RoboDK station: RK3 extrudy.rdk

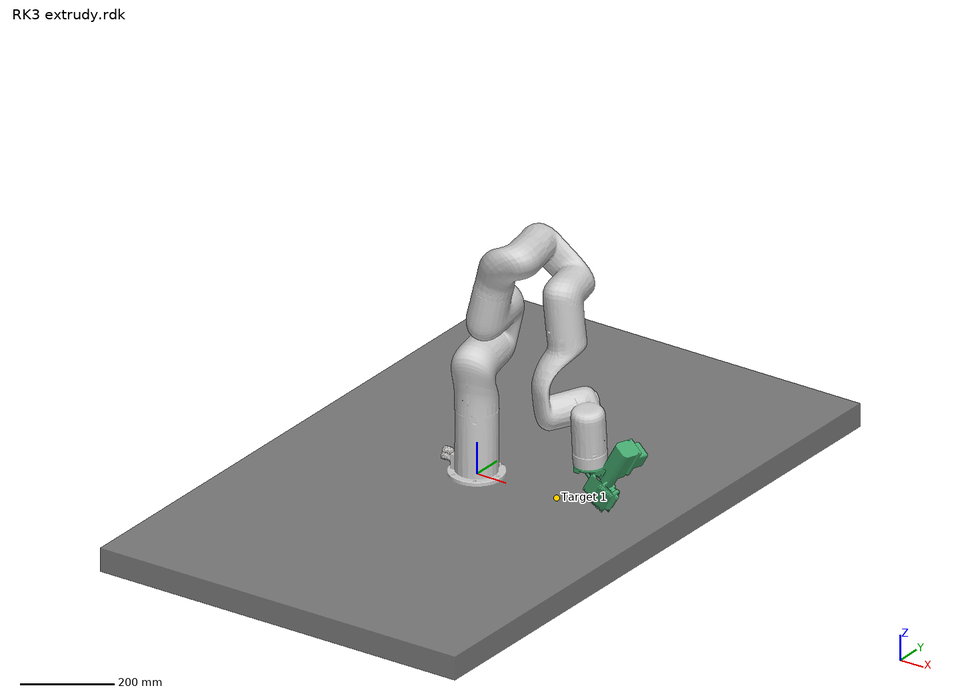
[picture v0: the station drawn from its stored meshes, robots at their saved joint values, targets as dots, program paths as lines]
Station RK3 extrudy (saved by RoboDK 5.5.0). Poses are relative to the parent item; angles as X-Y-Z fixed-axis rotations.
Station parameters (name, value as stored): CollisionFreePlanner, uFactory xArm6 11-16-2023 clayextruder, CollisionFreePlanner-Rob uFactory xArm6 11-16-2023 clayextruder
  - frame uFactory xArm6 Base at (0, 1000, 0) mm
    - robot uFactory xArm6 11-16-2023 clayextruder (model uFactory xArm6): 6 axes, payload 5 kg, reach 700 mm, repeatability 0.1 mm, weight 12.2 kg
        modified DH rows (alpha deg, a mm, theta deg, d mm): 0, 0, 0, 267; -90, 0, -79.35, 0; 0, 289.489, 79.35, 0; -90, 77.5, 0, 342.5; 90, 0, 0, 0; -90, 76, 0, 97
        joint limits [-360, -118, -225, -360, -81, -124] to [360, 120, 11, 360, 180, 110]; home [0, 0, 0, 0, 0, 0]; saved at [11.871, 11.935, -17.899, 43.294, 7.272, -31.184]
      - tool WASP extruder, TCP at (0, 0, 108) mm, rotated rx 0 ry -30.3 rz 0 deg, size 160.2 x 105.1 x 183.1 mm, geometry from uFactory xArm6 Base
  - frame uFactory xArm6 Base at (0, 1000, 0) mm
    - object table at (0, 0, 0) mm, rotated rx 90 ry 0 rz 90 deg, size 1500 x 55 x 920 mm, geometry from table.obj
    - target Target 1 (Cartesian target) at (207, 0, 0.5) mm, rotated rx -180 ry 30.3 rz 0 deg; joints [0, 0, 0, 0, 0, 0] of uFactory xArm6 11-16-2023 clayextruder
  - Python program Prog2 (listed below)

--- Python program Prog2 ---
# Type help("robodk.robolink") or help("robodk.robomath") for more information
# Press F5 to run the script
# Documentation: https://robodk.com/doc/en/RoboDK-API.html
# Reference:     https://robodk.com/doc/en/PythonAPI/robodk.html
# Note: It is not required to keep a copy of this file, your Python script is saved with your RDK project

# Forward and backwards compatible use of the RoboDK API:
# Remove these 2 lines to follow python programming guidelines
from robodk import *      # RoboDK API
from robolink import *    # Robot toolbox
# Link to RoboDK
# RDK = Robolink()

#generated with Grasshopper for Rhino
#Chris Morrey

import os
import sys
import time
import math

sys.path.append("C:\\Users\\morr0289\\Documents\\Github\\RobotArm\\Python\\")

from arm_sdk3.xarm.wrapper.xarm_api import XArmAPI
arm = XArmAPI('192.168.1.240')
id = 9
baudRate = 9600

if arm.warn_code != 0:
    arm.clean_warn()
if arm.error_code != 0:
    arm.clean_error()
time.sleep(2)

ret = arm.core.set_modbus_timeout(7)
print('set modbus timeout, ret = %d' % (ret[0]))
ret = arm.core.set_modbus_baudrate(baudRate)
print('set modbus baudrate, ret = %d' % (ret[0]))

time.sleep(1)
line = 102

def errors(returned):
    if returned == 1:
        print('1: uncleared error exists')
    elif returned == 23:
        print('23:modbus reply length error')
    elif returned == 20:
        print('20: wrong slave id')
    elif returned == 15:
        print('15: Modbus commands full')
    elif returned == 19:
        print('19: communication error')
    elif returned == 28:
        print('28: end module communication error')
    else:
        print('other error: ',returned)
    input=('clear errors? (y/n)')
    if input == 'y':
            arm.clean_error()
    else:
        print('error not cleared; quitting...')
        time.sleep(2)
        quit()
def sender(data_frame):
    global line
    global id
    #arm.clean_error()
    arm.set_state(state=0)
    code, digitals = arm.get_tgpio_digital()
    #while arm.connected and arm.error_code != 19 and arm.error_code != 28:
    if code == 0 and digitals[0] == 1:
        print ('extruder reports ready')
        ret = arm.getset_tgpio_modbus_data(data_frame,host_id=id)
        if ret[0] == 0:
            print('wrote ',data_frame[8],data_frame[9],data_frame[10])
            print('got back this: ',ret[1])
            print('line: ',line)
            line += 3
            time.sleep(.75)
    elif digitals [0] == 0:
        print('extruder reports not ready')
    elif code != 0:
        errors(ret[0])

arm.motion_enable(enable=True)
arm.set_mode(0)
arm.set_state(state=0)

arm.set_tcp_load(weight=0.91, center_of_gravity=[0,80,-40])
arm.set_tcp_offset([0,0,110,0,30.3,0], is_radian=False)
arm.set_collision_tool_model(22, x=40, y=40, z=110)

last_digitals = [-1, -1]

'''TGPIO for air solenoid---------------------------------------------
value = 0

    code = arm.set_cgpio_digital_output_function(i, value)
    print('set_cgpio_digital_output_function({}, {}), code={}'.format(i, value, code))
# Reset: 255
for i in range(4, 8):
    code = arm.set_cgpio_digital_output_function(i, 255)
    print('set_cgpio_digital_output_function({}, {}), code={}'.format(i, value, code))'''


arm.reset(wait=True)
if arm.warn_code != 0:
    arm.clean_warn()
if arm.error_code != 0:
    arm.clean_error()

while arm.connected and arm.error_code == 0:
#data is big-endian
    arm.set_position(x=272.50, y=-10.76, z=1.85, roll=180.0, pitch=-30.0, yaw=0.00, speed=30.00, is_radian=False, wait=True)
    datas = [0x09,0x10,0x00,0x00,0x00,0x04,0x08,0x00,0x15,0x00,0x06,0x00,0x01,0x00,0x65]
    sender(datas)
    arm.set_position(x=272.50, y=10.76, z=1.85, roll=180.0, pitch=-30.0, yaw=0.00, speed=30.00, is_radian=False, wait=True)
    datas = [0x09,0x10,0x00,0x00,0x00,0x04,0x08,0x00,0x05,0x00,0x06,0x00,0x01,0x00,0x68]
    sender(datas)
    arm.set_position(x=275.05, y=15.69, z=1.85, roll=180.0, pitch=-30.0, yaw=0.00, speed=30.00, is_radian=False, wait=True)
    datas = [0x09,0x10,0x00,0x00,0x00,0x04,0x08,0x00,0x1f,0x00,0x06,0x00,0x01,0x00,0x6b]
    sender(datas)
    arm.set_position(x=275.05, y=-15.69, z=1.85, roll=180.0, pitch=-30.0, yaw=0.00, speed=30.00, is_radian=False, wait=True)
    datas = [0x09,0x10,0x00,0x00,0x00,0x04,0x08,0x00,0x04,0x00,0x06,0x00,0x01,0x00,0x6e]
    sender(datas)
    arm.set_position(x=277.60, y=-19.35, z=1.85, roll=180.0, pitch=-30.0, yaw=0.00, speed=30.00, is_radian=False, wait=True)
    datas = [0x09,0x10,0x00,0x00,0x00,0x04,0x08,0x00,0x26,0x00,0x06,0x00,0x01,0x00,0x71]
    sender(datas)
    arm.set_position(x=277.60, y=19.35, z=1.85, roll=180.0, pitch=-30.0, yaw=0.00, speed=30.00, is_radian=False, wait=True)
    datas = [0x09,0x10,0x00,0x00,0x00,0x04,0x08,0x00,0x03,0x00,0x06,0x00,0x01,0x00,0x74]
    sender(datas)
    arm.set_position(x=280.15, y=22.36, z=1.85, roll=180.0, pitch=-30.0, yaw=0.00, speed=30.00, is_radian=False, wait=True)
    datas = [0x09,0x10,0x00,0x00,0x00,0x04,0x08,0x00,0x2c,0x00,0x06,0x00,0x01,0x00,0x77]
    sender(datas)
    arm.set_position(x=280.15, y=-22.36, z=1.85, roll=180.0, pitch=-30.0, yaw=0.00, speed=30.00, is_radian=False, wait=True)
    datas = [0x09,0x10,0x00,0x00,0x00,0x04,0x08,0x00,0x03,0x00,0x06,0x00,0x01,0x00,0x7a]
    sender(datas)
    arm.set_position(x=282.70, y=-24.96, z=1.85, roll=180.0, pitch=-30.0, yaw=0.00, speed=30.00, is_radian=False, wait=True)
    datas = [0x09,0x10,0x00,0x00,0x00,0x04,0x08,0x00,0x31,0x00,0x06,0x00,0x01,0x00,0x7d]
    sender(datas)
    arm.set_position(x=282.70, y=24.96, z=1.85, roll=180.0, pitch=-30.0, yaw=0.00, speed=30.00, is_radian=False, wait=True)
    datas = [0x09,0x10,0x00,0x00,0x00,0x04,0x08,0x00,0x03,0x00,0x06,0x00,0x01,0x00,0x80]
    sender(datas)
    arm.set_position(x=285.25, y=27.27, z=1.85, roll=180.0, pitch=-30.0, yaw=0.00, speed=30.00, is_radian=False, wait=True)
    datas = [0x09,0x10,0x00,0x00,0x00,0x04,0x08,0x00,0x36,0x00,0x06,0x00,0x01,0x00,0x83]
    sender(datas)
    arm.set_position(x=285.25, y=-27.27, z=1.85, roll=180.0, pitch=-30.0, yaw=0.00, speed=30.00, is_radian=False, wait=True)
    datas = [0x09,0x10,0x00,0x00,0x00,0x04,0x08,0x00,0x03,0x00,0x06,0x00,0x01,0x00,0x86]
    sender(datas)
    arm.set_position(x=287.80, y=-29.36, z=1.85, roll=180.0, pitch=-30.0, yaw=0.00, speed=30.00, is_radian=False, wait=True)
    datas = [0x09,0x10,0x00,0x00,0x00,0x04,0x08,0x00,0x3a,0x00,0x06,0x00,0x01,0x00,0x89]
    sender(datas)
    arm.set_position(x=287.80, y=29.36, z=1.85, roll=180.0, pitch=-30.0, yaw=0.00, speed=30.00, is_radian=False, wait=True)
    datas = [0x09,0x10,0x00,0x00,0x00,0x04,0x08,0x00,0x03,0x00,0x06,0x00,0x01,0x00,0x8c]
    sender(datas)
    arm.set_position(x=290.35, y=31.27, z=1.85, roll=180.0, pitch=-30.0, yaw=0.00, speed=30.00, is_radian=False, wait=True)
    datas = [0x09,0x10,0x00,0x00,0x00,0x04,0x08,0x00,0x3e,0x00,0x06,0x00,0x01,0x00,0x8f]
    sender(datas)
    arm.set_position(x=290.35, y=-31.27, z=1.85, roll=180.0, pitch=-30.0, yaw=0.00, speed=30.00, is_radian=False, wait=True)
    datas = [0x09,0x10,0x00,0x00,0x00,0x04,0x08,0x00,0x03,0x00,0x06,0x00,0x01,0x00,0x92]
    sender(datas)
    arm.set_position(x=292.90, y=-33.03, z=1.85, roll=180.0, pitch=-30.0, yaw=0.00, speed=30.00, is_radian=False, wait=True)
    datas = [0x09,0x10,0x00,0x00,0x00,0x04,0x08,0x00,0x42,0x00,0x06,0x00,0x01,0x00,0x95]
    sender(datas)
    arm.set_position(x=292.90, y=33.03, z=1.85, roll=180.0, pitch=-30.0, yaw=0.00, speed=30.00, is_radian=False, wait=True)
    datas = [0x09,0x10,0x00,0x00,0x00,0x04,0x08,0x00,0x03,0x00,0x06,0x00,0x01,0x00,0x98]
    sender(datas)
    arm.set_position(x=295.45, y=34.66, z=1.85, roll=180.0, pitch=-30.0, yaw=0.00, speed=30.00, is_radian=False, wait=True)
    datas = [0x09,0x10,0x00,0x00,0x00,0x04,0x08,0x00,0x45,0x00,0x06,0x00,0x01,0x00,0x9b]
    sender(datas)
    arm.set_position(x=295.45, y=-34.66, z=1.85, roll=180.0, pitch=-30.0, yaw=0.00, speed=30.00, is_radian=False, wait=True)
    datas = [0x09,0x10,0x00,0x00,0x00,0x04,0x08,0x00,0x02,0x00,0x06,0x00,0x01,0x00,0x9e]
    sender(datas)
    arm.set_position(x=298.00, y=-36.18, z=1.85, roll=180.0, pitch=-30.0, yaw=0.00, speed=30.00, is_radian=False, wait=True)
    datas = [0x09,0x10,0x00,0x00,0x00,0x04,0x08,0x00,0x48,0x00,0x06,0x00,0x01,0x00,0xa1]
    sender(datas)
    arm.set_position(x=298.00, y=36.18, z=1.85, roll=180.0, pitch=-30.0, yaw=0.00, speed=30.00, is_radian=False, wait=True)
    datas = [0x09,0x10,0x00,0x00,0x00,0x04,0x08,0x00,0x02,0x00,0x06,0x00,0x01,0x00,0xa4]
    sender(datas)
    arm.set_position(x=300.55, y=37.60, z=1.85, roll=180.0, pitch=-30.0, yaw=0.00, speed=30.00, is_radian=False, wait=True)
    datas = [0x09,0x10,0x00,0x00,0x00,0x04,0x08,0x00,0x4b,0x00,0x06,0x00,0x01,0x00,0xa7]
    sender(datas)
    arm.set_position(x=300.55, y=-37.60, z=1.85, roll=180.0, pitch=-30.0, yaw=0.00, speed=30.00, is_radian=False, wait=True)
    datas = [0x09,0x10,0x00,0x00,0x00,0x04,0x08,0x00,0x02,0x00,0x06,0x00,0x01,0x00,0xaa]
    sender(datas)
    arm.set_position(x=303.10, y=-38.95, z=1.85, roll=180.0, pitch=-30.0, yaw=0.00, speed=30.00, is_radian=False, wait=True)
    datas = [0x09,0x10,0x00,0x00,0x00,0x04,0x08,0x00,0x4d,0x00,0x06,0x00,0x01,0x00,0xad]
    sender(datas)
    arm.set_position(x=303.10, y=38.95, z=1.85, roll=180.0, pitch=-30.0, yaw=0.00, speed=30.00, is_radian=False, wait=True)
    datas = [0x09,0x10,0x00,0x00,0x00,0x04,0x08,0x00,0x02,0x00,0x06,0x00,0x01,0x00,0xb0]
    sender(datas)
    arm.set_position(x=305.65, y=40.21, z=1.85, roll=180.0, pitch=-30.0, yaw=0.00, speed=30.00, is_radian=False, wait=True)
    datas = [0x09,0x10,0x00,0x00,0x00,0x04,0x08,0x00,0x50,0x00,0x06,0x00,0x01,0x00,0xb3]
    sender(datas)
    arm.set_position(x=305.65, y=-40.21, z=1.85, roll=180.0, pitch=-30.0, yaw=0.00, speed=30.00, is_radian=False, wait=True)
    datas = [0x09,0x10,0x00,0x00,0x00,0x04,0x08,0x00,0x02,0x00,0x06,0x00,0x01,0x00,0xb6]
    sender(datas)
    arm.set_position(x=308.20, y=-41.40, z=1.85, roll=180.0, pitch=-30.0, yaw=0.00, speed=30.00, is_radian=False, wait=True)
    datas = [0x09,0x10,0x00,0x00,0x00,0x04,0x08,0x00,0x52,0x00,0x06,0x00,0x01,0x00,0xb9]
    sender(datas)
    arm.set_position(x=308.20, y=41.40, z=1.85, roll=180.0, pitch=-30.0, yaw=0.00, speed=30.00, is_radian=False, wait=True)
    datas = [0x09,0x10,0x00,0x00,0x00,0x04,0x08,0x00,0x02,0x00,0x06,0x00,0x01,0x00,0xbc]
    sender(datas)
    arm.set_position(x=310.75, y=42.53, z=1.85, roll=180.0, pitch=-30.0, yaw=0.00, speed=30.00, is_radian=False, wait=True)
    datas = [0x09,0x10,0x00,0x00,0x00,0x04,0x08,0x00,0x55,0x00,0x06,0x00,0x01,0x00,0xbf]
    sender(datas)
    arm.set_position(x=310.75, y=-42.53, z=1.85, roll=180.0, pitch=-30.0, yaw=0.00, speed=30.00, is_radian=False, wait=True)
    datas = [0x09,0x10,0x00,0x00,0x00,0x04,0x08,0x00,0x02,0x00,0x06,0x00,0x01,0x00,0xc2]
    sender(datas)
    arm.set_position(x=313.30, y=-43.60, z=1.85, roll=180.0, pitch=-30.0, yaw=0.00, speed=30.00, is_radian=False, wait=True)
    datas = [0x09,0x10,0x00,0x00,0x00,0x04,0x08,0x00,0x57,0x00,0x06,0x00,0x01,0x00,0xc5]
    sender(datas)
    arm.set_position(x=313.30, y=43.60, z=1.85, roll=180.0, pitch=-30.0, yaw=0.00, speed=30.00, is_radian=False, wait=True)
    datas = [0x09,0x10,0x00,0x00,0x00,0x04,0x08,0x00,0x02,0x00,0x06,0x00,0x01,0x00,0xc8]
    sender(datas)
    arm.set_position(x=315.85, y=44.62, z=1.85, roll=180.0, pitch=-30.0, yaw=0.00, speed=30.00, is_radian=False, wait=True)
    datas = [0x09,0x10,0x00,0x00,0x00,0x04,0x08,0x00,0x59,0x00,0x06,0x00,0x01,0x00,0xcb]
    sender(datas)
    arm.set_position(x=315.85, y=-44.62, z=1.85, roll=180.0, pitch=-30.0, yaw=0.00, speed=30.00, is_radian=False, wait=True)
    datas = [0x09,0x10,0x00,0x00,0x00,0x04,0x08,0x00,0x02,0x00,0x06,0x00,0x01,0x00,0xce]
    sender(datas)
    arm.set_position(x=318.40, y=-45.58, z=1.85, roll=180.0, pitch=-30.0, yaw=0.00, speed=30.00, is_radian=False, wait=True)
    datas = [0x09,0x10,0x00,0x00,0x00,0x04,0x08,0x00,0x5b,0x00,0x06,0x00,0x01,0x00,0xd1]
    sender(datas)
    arm.set_position(x=318.40, y=45.58, z=1.85, roll=180.0, pitch=-30.0, yaw=0.00, speed=30.00, is_radian=False, wait=True)
    datas = [0x09,0x10,0x00,0x00,0x00,0x04,0x08,0x00,0x02,0x00,0x06,0x00,0x01,0x00,0xd4]
    sender(datas)
    arm.set_position(x=320.95, y=46.49, z=1.85, roll=180.0, pitch=-30.0, yaw=0.00, speed=30.00, is_radian=False, wait=True)
    datas = [0x09,0x10,0x00,0x00,0x00,0x04,0x08,0x00,0x5c,0x00,0x06,0x00,0x01,0x00,0xd7]
    sender(datas)
    arm.set_position(x=320.95, y=-46.49, z=1.85, roll=180.0, pitch=-30.0, yaw=0.00, speed=30.00, is_radian=False, wait=True)
    datas = [0x09,0x10,0x00,0x00,0x00,0x04,0x08,0x00,0x02,0x00,0x06,0x00,0x01,0x00,0xda]
    sender(datas)
    arm.set_position(x=323.50, y=-47.36, z=1.85, roll=180.0, pitch=-30.0, yaw=0.00, speed=30.00, is_radian=False, wait=True)
    datas = [0x09,0x10,0x00,0x00,0x00,0x04,0x08,0x00,0x5e,0x00,0x06,0x00,0x01,0x00,0xdd]
    sender(datas)
    arm.set_position(x=323.50, y=47.36, z=1.85, roll=180.0, pitch=-30.0, yaw=0.00, speed=30.00, is_radian=False, wait=True)
    datas = [0x09,0x10,0x00,0x00,0x00,0x04,0x08,0x00,0x02,0x00,0x06,0x00,0x01,0x00,0xe0]
    sender(datas)
    arm.set_position(x=326.05, y=48.19, z=1.85, roll=180.0, pitch=-30.0, yaw=0.00, speed=30.00, is_radian=False, wait=True)
    datas = [0x09,0x10,0x00,0x00,0x00,0x04,0x08,0x00,0x60,0x00,0x06,0x00,0x01,0x00,0xe3]
    sender(datas)
    arm.set_position(x=326.05, y=-48.19, z=1.85, roll=180.0, pitch=-30.0, yaw=0.00, speed=30.00, is_radian=False, wait=True)
    datas = [0x09,0x10,0x00,0x00,0x00,0x04,0x08,0x00,0x02,0x00,0x06,0x00,0x01,0x00,0xe6]
    sender(datas)
    arm.set_position(x=328.60, y=-48.97, z=1.85, roll=180.0, pitch=-30.0, yaw=0.00, speed=30.00, is_radian=False, wait=True)
    datas = [0x09,0x10,0x00,0x00,0x00,0x04,0x08,0x00,0x61,0x00,0x06,0x00,0x01,0x00,0xe9]
    sender(datas)
    arm.set_position(x=328.60, y=48.97, z=1.85, roll=180.0, pitch=-30.0, yaw=0.00, speed=30.00, is_radian=False, wait=True)
    datas = [0x09,0x10,0x00,0x00,0x00,0x04,0x08,0x00,0x02,0x00,0x06,0x00,0x01,0x00,0xec]
    sender(datas)
    arm.set_position(x=331.15, y=49.72, z=1.85, roll=180.0, pitch=-30.0, yaw=0.00, speed=30.00, is_radian=False, wait=True)
    datas = [0x09,0x10,0x00,0x00,0x00,0x04,0x08,0x00,0x63,0x00,0x06,0x00,0x01,0x00,0xef]
    sender(datas)
    arm.set_position(x=331.15, y=-49.72, z=1.85, roll=180.0, pitch=-30.0, yaw=0.00, speed=30.00, is_radian=False, wait=True)
    datas = [0x09,0x10,0x00,0x00,0x00,0x04,0x08,0x00,0x02,0x00,0x06,0x00,0x01,0x00,0xf2]
    sender(datas)
    arm.set_position(x=333.70, y=-50.43, z=1.85, roll=180.0, pitch=-30.0, yaw=0.00, speed=30.00, is_radian=False, wait=True)
    datas = [0x09,0x10,0x00,0x00,0x00,0x04,0x08,0x00,0x64,0x00,0x06,0x00,0x01,0x00,0xf5]
    sender(datas)
    arm.set_position(x=333.70, y=50.43, z=1.85, roll=180.0, pitch=-30.0, yaw=0.00, speed=30.00, is_radian=False, wait=True)
    datas = [0x09,0x10,0x00,0x00,0x00,0x04,0x08,0x00,0x02,0x00,0x06,0x00,0x01,0x00,0xf8]
    sender(datas)
    arm.set_position(x=336.25, y=51.10, z=1.85, roll=180.0, pitch=-30.0, yaw=0.00, speed=30.00, is_radian=False, wait=True)
    datas = [0x09,0x10,0x00,0x00,0x00,0x04,0x08,0x00,0x66,0x00,0x06,0x00,0x01,0x00,0xfb]
    sender(datas)
    arm.set_position(x=336.25, y=-51.10, z=1.85, roll=180.0, pitch=-30.0, yaw=0.00, speed=30.00, is_radian=False, wait=True)
    datas = [0x09,0x10,0x00,0x00,0x00,0x04,0x08,0x00,0x02,0x00,0x06,0x00,0x01,0x00,0xfe]
    sender(datas)
    arm.set_position(x=338.80, y=-51.74, z=1.85, roll=180.0, pitch=-30.0, yaw=0.00, speed=30.00, is_radian=False, wait=True)
    datas = [0x09,0x10,0x00,0x00,0x00,0x04,0x08,0x00,0x67,0x00,0x06,0x00,0x01,0x01,0x01]
    sender(datas)
    arm.set_position(x=338.80, y=51.74, z=1.85, roll=180.0, pitch=-30.0, yaw=0.00, speed=30.00, is_radian=False, wait=True)
    datas = [0x09,0x10,0x00,0x00,0x00,0x04,0x08,0x00,0x02,0x00,0x06,0x00,0x01,0x01,0x04]
    sender(datas)
    arm.set_position(x=341.35, y=52.34, z=1.85, roll=180.0, pitch=-30.0, yaw=0.00, speed=30.00, is_radian=False, wait=True)
    datas = [0x09,0x10,0x00,0x00,0x00,0x04,0x08,0x00,0x68,0x00,0x06,0x00,0x01,0x01,0x07]
    sender(datas)
    arm.set_position(x=341.35, y=-52.34, z=1.85, roll=180.0, pitch=-30.0, yaw=0.00, speed=30.00, is_radian=False, wait=True)
    datas = [0x09,0x10,0x00,0x00,0x00,0x04,0x08,0x00,0x02,0x00,0x06,0x00,0x01,0x01,0x0a]
    sender(datas)
    arm.set_position(x=343.90, y=-52.91, z=1.85, roll=180.0, pitch=-30.0, yaw=0.00, speed=30.00, is_radian=False, wait=True)
    datas = [0x09,0x10,0x00,0x00,0x00,0x04,0x08,0x00,0x69,0x00,0x06,0x00,0x01,0x01,0x0d]
    sender(datas)
    arm.set_position(x=343.90, y=52.91, z=1.85, roll=180.0, pitch=-30.0, yaw=0.00, speed=30.00, is_radian=False, wait=True)
    datas = [0x09,0x10,0x00,0x00,0x00,0x04,0x08,0x00,0x02,0x00,0x06,0x00,0x01,0x01,0x10]
    sender(datas)
    arm.set_position(x=346.45, y=53.46, z=1.85, roll=180.0, pitch=-30.0, yaw=0.00, speed=30.00, is_radian=False, wait=True)
    datas = [0x09,0x10,0x00,0x00,0x00,0x04,0x08,0x00,0x6a,0x00,0x06,0x00,0x01,0x01,0x13]
    sender(datas)
    arm.set_position(x=346.45, y=-53.46, z=1.85, roll=180.0, pitch=-30.0, yaw=0.00, speed=30.00, is_radian=False, wait=True)
    datas = [0x09,0x10,0x00,0x00,0x00,0x04,0x08,0x00,0x02,0x00,0x06,0x00,0x01,0x01,0x16]
    sender(datas)
    arm.set_position(x=349.00, y=-53.97, z=1.85, roll=180.0, pitch=-30.0, yaw=0.00, speed=30.00, is_radian=False, wait=True)
    datas = [0x09,0x10,0x00,0x00,0x00,0x04,0x08,0x00,0x6b,0x00,0x06,0x00,0x01,0x01,0x19]
    sender(datas)
    arm.set_position(x=349.00, y=53.97, z=1.85, roll=180.0, pitch=-30.0, yaw=0.00, speed=30.00, is_radian=False, wait=True)
    datas = [0x09,0x10,0x00,0x00,0x00,0x04,0x08,0x00,0x02,0x00,0x06,0x00,0x01,0x01,0x1c]
    sender(datas)
    arm.set_position(x=351.55, y=54.45, z=1.85, roll=180.0, pitch=-30.0, yaw=0.00, speed=30.00, is_radian=False, wait=True)
    datas = [0x09,0x10,0x00,0x00,0x00,0x04,0x08,0x00,0x6c,0x00,0x06,0x00,0x01,0x01,0x1f]
    sender(datas)
    arm.set_position(x=351.55, y=-54.45, z=1.85, roll=180.0, pitch=-30.0, yaw=0.00, speed=30.00, is_radian=False, wait=True)
    datas = [0x09,0x10,0x00,0x00,0x00,0x04,0x08,0x00,0x02,0x00,0x06,0x00,0x01,0x01,0x22]
    sender(datas)
    arm.set_position(x=354.10, y=-54.90, z=1.85, roll=180.0, pitch=-30.0, yaw=0.00, speed=30.00, is_radian=False, wait=True)
    datas = [0x09,0x10,0x00,0x00,0x00,0x04,0x08,0x00,0x6d,0x00,0x06,0x00,0x01,0x01,0x25]
    sender(datas)
    arm.set_position(x=354.10, y=54.90, z=1.85, roll=180.0, pitch=-30.0, yaw=0.00, speed=30.00, is_radian=False, wait=True)
    datas = [0x09,0x10,0x00,0x00,0x00,0x04,0x08,0x00,0x02,0x00,0x06,0x00,0x01,0x01,0x28]
    sender(datas)
    arm.set_position(x=356.65, y=55.33, z=1.85, roll=180.0, pitch=-30.0, yaw=0.00, speed=30.00, is_radian=False, wait=True)
    datas = [0x09,0x10,0x00,0x00,0x00,0x04,0x08,0x00,0x6e,0x00,0x06,0x00,0x01,0x01,0x2b]
    sender(datas)
#finish up:
datas =[0x09,0x10,0x00,0x03,0x00,0x01,0x02,0x00,0x01]
sender(datas)
time.sleep(2)
arm.reset(wait=True)
arm.disconnect()
